FUNCTION_BLOCK FB_CalcXY
(* Berechnung des a und b Wertes für die Linearisierung Y=ax+b *)
VAR_INPUT
     Dev : POINTER TO DUT_Device;
END_VAR
VAR_OUTPUT

END_VAR 
VAR

END_VAR

(* prevent Div By Zero *)

Dev^.dFakt_A := 1;
Dev^.dSmd_B := 0;

IF (Dev^.rIN_HI - Dev^.rIN_LO) = 0 THEN
     RETURN;
END_IF

Dev^.dFakt_A :=  UINT_TO_REAL(Dev^.nOUT_HI - Dev^.nOUT_LO ) / (Dev^.rIN_HI - Dev^.rIN_LO);
Dev^.dSmd_B := Dev^.nOUT_LO - (Dev^.rIN_LO * Dev^.dFakt_A);

END_FUNCTION_BLOCK

(* stored: Version 1.1.0.1, ProductVersion 3.1.4024.3
   POU FB_CalcXY: Id {3f5d1098-50c2-4f0c-9487-99b4e55b7df3}, SpecialFunc None *)
